TYPE ST_InsulationMonitor_get :
STRUCT
	b_Enabled							: BOOL;	
	b_PENlinkNotDetected				: BOOL;
	b_Warning							: BOOL;
END_STRUCT
END_TYPE

(* stored: Version 1.1.0.1, ProductVersion 3.1.4024.12
   DUT ST_InsulationMonitor_get: Id {f03fda51-285c-4fb6-9458-9a5320accc13} *)
